// TIA Portal V19 export
FUNCTION "DATE&TIMES" : Void   // FC9, LAD
{ S7_Optimized_Access := 'TRUE' }
// stored: SetENOAutomatically false
BEGIN

REGION Network 1
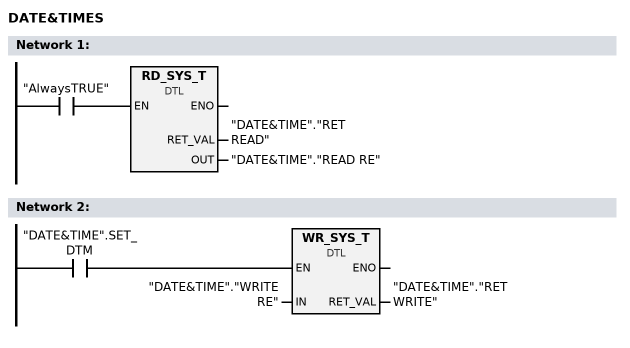
   RUNG wire#powerrail
      Contact( "AlwaysTRUE" )
      { S7_Templates := "date_type := DTL" } RD_SYS_T(RET_VAL => "DATE&TIME"."RET READ", OUT => "DATE&TIME"."READ RE")
   END_RUNG
   // the same network as SCL:
   IF "AlwaysTRUE" THEN "DATE&TIME"."RET READ" := RD_SYS_T(OUT => "DATE&TIME"."READ RE"); END_IF;
END_REGION

REGION Network 2
   RUNG wire#powerrail
      Contact( "DATE&TIME".SET_DTM )
      { S7_Templates := "date_type := DTL" } WR_SYS_T(IN := "DATE&TIME"."WRITE RE", RET_VAL => "DATE&TIME"."RET WRITE")
   END_RUNG
   // the same network as SCL:
   IF "DATE&TIME".SET_DTM THEN "DATE&TIME"."RET WRITE" := WR_SYS_T(IN := "DATE&TIME"."WRITE RE"); END_IF;
END_REGION
END_FUNCTION
